TYPE CmpConvBreakStopGroup :
STRUCT
	Framework: Framework;
	ConvRunning: ARRAY[1..cBreakStopGroupMaxInstance] OF BOOL;
	LowerStopReq: ARRAY[1..cBreakStopGroupMaxInstance] OF BOOL;
	Config: CmpConvBreakStopGroupConfig;
END_STRUCT
END_TYPE

(* stored: Version 1.1.0.1, ProductVersion 3.1.4024.6
   DUT CmpConvBreakStopGroup: Id {f6a66bb0-5195-46be-afa9-89697ece1c58} *)
